// TIA Portal V17 export
// export: Created 2025-06-26T06:49:17.9536247Z, ExportSetting WithDefaults, DisplayName Totally Integrated Automation Portal, DisplayVersion V17 Update 8, DisplayName TIA Portal Openness, DisplayVersion V17 Update 8, DisplayName TIA Portal Version Control Interface, DisplayVersion V17, DisplayName STEP 7 Professional, DisplayVersion V17 Update 8, DisplayName STEP 7 Safety, DisplayVersion V17 Update 6, DisplayName WinCC Advanced, DisplayVersion V17 Update 8
FUNCTION "ProcessModuleCalculations" : Void   // FC16, FBD
{ S7_Optimized_Access := 'TRUE' }
VERSION : 0.1
// stored: AutoNumber true, IsIECCheckEnabled false, SetENOAutomatically false, UDAEnableTagReadback false
   VAR_TEMP
      T_Evaporation_LP : Real;
      T_Condense_HP : Real;
   END_VAR
   VAR_TEMP   // added for the SCL form of the ladder/FBD networks
      _w1 : Bool;
   END_VAR
BEGIN

REGION Network 1: Evaporator discharge pressure mean
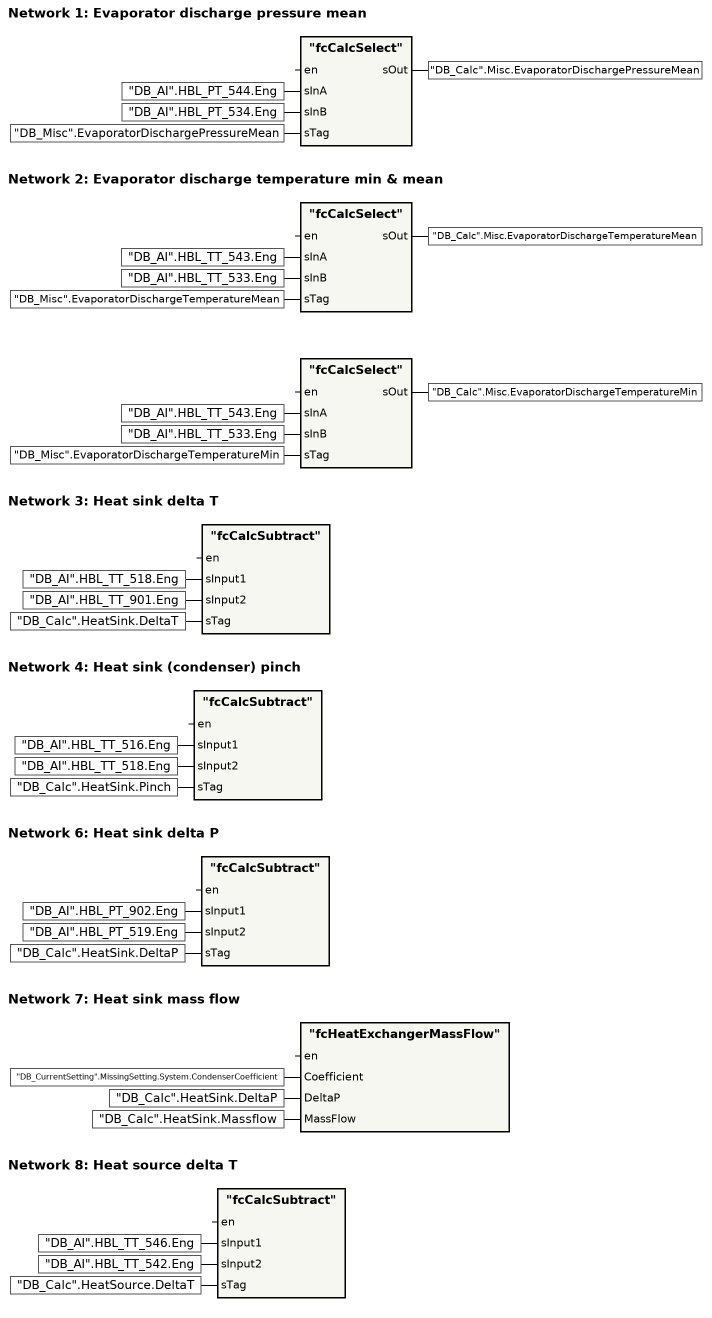
   "fcCalcSelect"(sInA := "DB_AI".HBL_PT_544.Eng,
                  sInB := "DB_AI".HBL_PT_534.Eng,
                  sTag := "DB_Misc".EvaporatorDischargePressureMean,
                  sOut => "DB_Calc".Misc.EvaporatorDischargePressureMean);
END_REGION

REGION Network 2: Evaporator discharge temperature min & mean
   "fcCalcSelect"(sInA := "DB_AI".HBL_TT_543.Eng,
                  sInB := "DB_AI".HBL_TT_533.Eng,
                  sTag := "DB_Misc".EvaporatorDischargeTemperatureMean,
                  sOut => "DB_Calc".Misc.EvaporatorDischargeTemperatureMean);
   "fcCalcSelect"(sInA := "DB_AI".HBL_TT_543.Eng,
                  sInB := "DB_AI".HBL_TT_533.Eng,
                  sTag := "DB_Misc".EvaporatorDischargeTemperatureMin,
                  sOut => "DB_Calc".Misc.EvaporatorDischargeTemperatureMin);
END_REGION

REGION Network 3: Heat sink delta T
   // Temperature rise (positive)
   "fcCalcSubtract"(sInput1 := "DB_AI".HBL_TT_518.Eng,
                    sInput2 := "DB_AI".HBL_TT_901.Eng,
                    sTag := "DB_Calc".HeatSink.DeltaT);
END_REGION

REGION Network 4: Heat sink (condenser) pinch
   // Pinch feed flow = Condenser suction temperature - Heat sink discharge temperature
   "fcCalcSubtract"(sInput1 := "DB_AI".HBL_TT_516.Eng,
                    sInput2 := "DB_AI".HBL_TT_518.Eng,
                    sTag := "DB_Calc".HeatSink.Pinch);
END_REGION

REGION Network 5: Heat sink heat rate
END_REGION

REGION Network 6: Heat sink delta P
   // Estimated from pressure drop across the condenser
   "fcCalcSubtract"(sInput1 := "DB_AI".HBL_PT_902.Eng,
                    sInput2 := "DB_AI".HBL_PT_519.Eng,
                    sTag := "DB_Calc".HeatSink.DeltaP);
END_REGION

REGION Network 7: Heat sink mass flow
   "fcHeatExchangerMassFlow"(Coefficient := "DB_CurrentSetting".MissingSetting.System.CondenserCoefficient,
                           DeltaP := "DB_Calc".HeatSink.DeltaP,
                           MassFlow := "DB_Calc".HeatSink.Massflow);
END_REGION

REGION Network 8: Heat source delta T
   // Temperature drop (positive)
   "fcCalcSubtract"(sInput1 := "DB_AI".HBL_TT_546.Eng,
                    sInput2 := "DB_AI".HBL_TT_542.Eng,
                    sTag := "DB_Calc".HeatSource.DeltaT);
END_REGION

REGION Network 9: Heat source pinch (evaporator)
   // Pinch return flow = Heat Source discharge temperature - Evaporation temperature
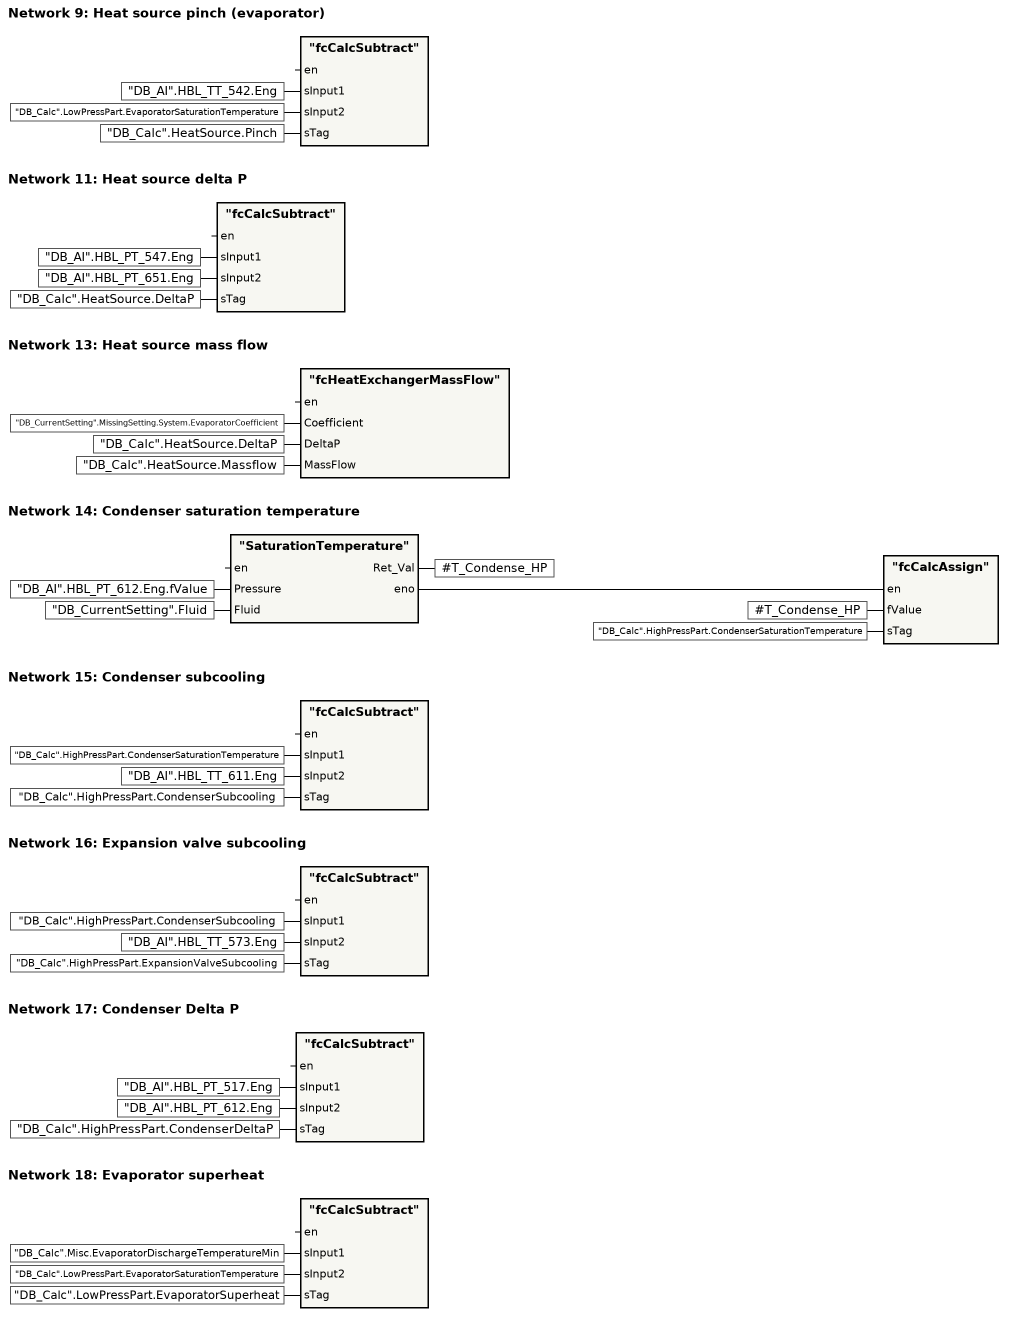
   "fcCalcSubtract"(sInput1 := "DB_AI".HBL_TT_542.Eng,
                    sInput2 := "DB_Calc".LowPressPart.EvaporatorSaturationTemperature,
                    sTag := "DB_Calc".HeatSource.Pinch);
END_REGION

REGION Network 10: Heat source heat rate
END_REGION

REGION Network 11: Heat source delta P
   // ##Note: this may not make a lot of sense. PT-547 is steam pressure, PT-651 is condensate pressure
   "fcCalcSubtract"(sInput1 := "DB_AI".HBL_PT_547.Eng,
                    sInput2 := "DB_AI".HBL_PT_651.Eng,
                    sTag := "DB_Calc".HeatSource.DeltaP);
END_REGION

REGION Network 12: Heat source temperature rate of change
   // in Calculations (FB42) as it requires static variables
END_REGION

REGION Network 13: Heat source mass flow
   "fcHeatExchangerMassFlow"(Coefficient := "DB_CurrentSetting".MissingSetting.System.EvaporatorCoefficient,
                           DeltaP := "DB_Calc".HeatSource.DeltaP,
                           MassFlow := "DB_Calc".HeatSource.Massflow);
END_REGION

REGION Network 14: Condenser saturation temperature
   #T_Condense_HP := "SaturationTemperature"(Pressure := "DB_AI".HBL_PT_612.Eng.fValue,
                           Fluid := "DB_CurrentSetting".Fluid,
                           ENO => #_w1);
   IF #_w1 THEN
       "fcCalcAssign"(fValue := #T_Condense_HP, sTag := "DB_Calc".HighPressPart.CondenserSaturationTemperature);
   END_IF;
END_REGION

REGION Network 15: Condenser subcooling
   "fcCalcSubtract"(sInput1 := "DB_Calc".HighPressPart.CondenserSaturationTemperature,
                    sInput2 := "DB_AI".HBL_TT_611.Eng,
                    sTag := "DB_Calc".HighPressPart.CondenserSubcooling);
END_REGION

REGION Network 16: Expansion valve subcooling
   "fcCalcSubtract"(sInput1 := "DB_Calc".HighPressPart.CondenserSubcooling,
                    sInput2 := "DB_AI".HBL_TT_573.Eng,
                    sTag := "DB_Calc".HighPressPart.ExpansionValveSubcooling);
END_REGION

REGION Network 17: Condenser Delta P
   "fcCalcSubtract"(sInput1 := "DB_AI".HBL_PT_517.Eng,
                    sInput2 := "DB_AI".HBL_PT_612.Eng,
                    sTag := "DB_Calc".HighPressPart.CondenserDeltaP);
END_REGION

REGION Network 18: Evaporator superheat
   "fcCalcSubtract"(sInput1 := "DB_Calc".Misc.EvaporatorDischargeTemperatureMin,
                    sInput2 := "DB_Calc".LowPressPart.EvaporatorSaturationTemperature,
                    sTag := "DB_Calc".LowPressPart.EvaporatorSuperheat);
END_REGION

REGION Network 19: Evaporator saturation temperature
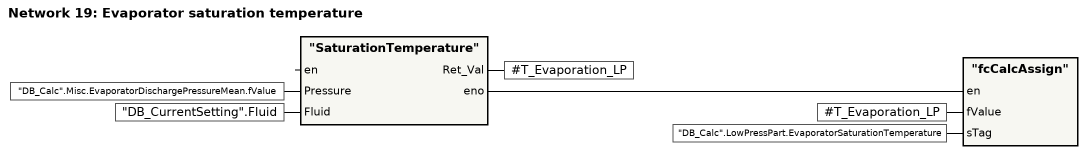
   #T_Evaporation_LP := "SaturationTemperature"(Pressure := "DB_Calc".Misc.EvaporatorDischargePressureMean.fValue,
                           Fluid := "DB_CurrentSetting".Fluid,
                           ENO => #_w1);
   IF #_w1 THEN
       "fcCalcAssign"(fValue := #T_Evaporation_LP, sTag := "DB_Calc".LowPressPart.EvaporatorSaturationTemperature);
   END_IF;
END_REGION
END_FUNCTION
